// TwinCAT 3 PLC project PLC
// ProgramVersion: 3.1.4022.1
// libraries:
//   Tc2_Standard, * (Beckhoff Automation GmbH)
//   Tc2_System, * (Beckhoff Automation GmbH)
//   Tc3_EventLogger, * (Beckhoff Automation GmbH)
//   Tc3_Module, * (Beckhoff Automation GmbH)
//   Tc3_JsonXml,3.3.4.0,Beckhoff Automation GmbH
// project tree:
//   DUTs/ ST_AI.TcDUT, ST_Led.TcDUT, ST_Values_LineChart.TcDUT
//   / GlobalTextList.TcGTLO, PlcTask.TcTTO
//   GVLs/ HMI.TcGVL
//   POUs/ CHART.TcPOU, FB_Blink.TcPOU, FB_LineChart.TcPOU, MAIN.TcPOU, SCOPE.TcPOU
//   POUs/Motor/ FB_Motor.TcPOU, ST_MotorParam.TcDUT
//   POUs/Valve/ FB_Valve.TcPOU, ST_ValveParam.TcDUT
// real-time tasks:
//   TASK PlcTask: cycle T#10ms, priority 20, ADS port 350

CONFIGURATION PLC
    RESOURCE PLC ON TwinCAT3
        TASK PlcTask(INTERVAL := T#10ms, PRIORITY := 20);
        PROGRAM MAIN WITH PlcTask : MAIN;
    END_RESOURCE
END_CONFIGURATION

// ---- DUTs/ST_AI.TcDUT
TYPE ST_AI :
STRUCT
ID: STRING;
Measure:REAL;
Low_Range:REAL;
High_Range:REAL;
Decimals:INT;
Unit:STRING;
Alarmtype:INT;
LowLimit: REAL;
LowDelay:DINT;
LowAlarm:BOOL;
HighLimit: REAL;
HighDelay:DINT;
HighAlarm:BOOL;
Sensortype:INT;
ShortCircuitAlarm:BOOL;
BrokenWireAlarm:BOOL;
Offset:REAL;
ManualValue:REAL;
ManualControl:INT;
END_STRUCT
END_TYPE

// ---- DUTs/ST_Led.TcDUT
TYPE ST_Led :
STRUCT
	sName 		: STRING;
	bControl	: BOOL;
	bStatus 	: BOOL;
	nValue		: REAL;
END_STRUCT
END_TYPE

// ---- DUTs/ST_Values_LineChart.TcDUT
TYPE ST_Values_LineChart :
STRUCT
	x:LREAL;
	y:LREAL;

END_STRUCT
END_TYPE

// ---- POUs/Motor/ST_MotorParam.TcDUT
TYPE ST_MotorParam :
STRUCT
	Unit : STRING;
	Set : INT;
	P: UINT;
	I: UINT;
	D: UINT;
END_STRUCT
END_TYPE

// ---- POUs/Valve/ST_ValveParam.TcDUT
TYPE ST_ValveParam :
STRUCT
	Unit : STRING;
	Set : INT;
	P: UINT;
	I: UINT;
	D: UINT;
END_STRUCT
END_TYPE

// ---- GVLs/HMI.TcGVL
{attribute 'qualified_only'}
VAR_GLOBAL
	bEnableLed	: BOOL;
	bLedStatus	: BOOL;
	stAi		: ST_AI;
	arrStLeds	: ARRAY[1..NUM_OF_LEDS] OF ST_Led := 
	[
		(sName := 'Led #01'),
		(sName := 'Led #02'),
		(sName := 'Led #03'),
		(sName := 'Led #04'),
		(sName := 'Led #05'),
		(sName := 'Led #06'),
		(sName := 'Led #07'),
		(sName := 'Led #08'),
		(sName := 'Led #09'),
		(sName := 'Led #10')
	];
	arrPersons	: ARRAY [1..NUM_OF_PERSONS] OF STRING := 
	[
		'Person1',
		'Person2',
		'Person3',
		'Person4',
		'Person5',
		'Person6',
		'Person7',
		'Person8',
		'Person9',
		'Person10'
	];
	SineVerySlow	: LREAL;
END_VAR

VAR_GLOBAL CONSTANT
	NUM_OF_LEDS : INT := 10;	
	NUM_OF_PERSONS : INT := 10;
END_VAR

// ---- POUs/MAIN.TcPOU
PROGRAM MAIN
VAR
	fbBlink		: FB_Blink;
	arrFbBlink 	: ARRAY [1..HMI.NUM_OF_LEDS] OF FB_Blink;
	i: INT;
	a: INT;
	b: INT := 1000;
	asdf: INT;
	stAi: INT;
	adfsaa: UINT;
	bInitAlarms: BOOL;
	sString : STRING := '{"color": "rgba(255,191,127,1)"}';
	
	fbEventLogger : FB_TcEventLogger;
	fbAlarm01 : FB_TcAlarm;
	fbMessage01 : FB_TcMessage;
	bTriggerAlarm01 : BOOL;
	bConfirmAlarm01 : BOOL;
	bClearAlarm01	: BOOL;
	
	stLed : REFERENCE TO ST_LED;
	stLedInstance : ST_LED;
	
	fbValve: FB_Valve;
	fbMotor: FB_Motor;
	LOGSTUFF: BOOL;
	asd: DINT;
END_VAR


// Yksittäisen FB:n kutsuminen
fbBlink(
	i_bEnable:= HMI.bEnableLed, 
	i_tTime := T#1S, 
	O_bOut=> hmi.bLedStatus
); 

// Taulukossa olevien FB:iden kutsuminen
FOR i := 1 TO HMI.NUM_OF_LEDS DO
	arrFbBlink[i]
	(
		i_sName 	:= HMI.arrStLeds[i].sName,
		i_bEnable 	:= HMI.arrStLeds[i].bControl,
		o_bOut		=> HMI.arrStLeds[i].bStatus
	);
END_FOR

SCOPE();

asdf := SIZEOF(HMI.stAi);
adfsaa := SIZEOF(HMI.arrStLeds[1]);


IF (NOT bInitAlarms) THEN
	bInitAlarms:=TRUE;
	fbAlarm01.CreateEx(TC_EVENTS.AlarmsClass.Alarm01,TRUE,0);
	fbMessage01.CreateEx(TC_EVENTS.AlarmsClass.Message01, 0);
END_IF

IF (bTriggerAlarm01) THEN
	fbAlarm01.Raise(0);
	bTriggerAlarm01 := FALSE;
END_IF

IF (bConfirmAlarm01) THEN
	fbAlarm01.Confirm(0);
	bConfirmAlarm01:= FALSE;
END_IF

IF (bClearAlarm01) THEN
	fbAlarm01.Clear(0,TRUE);
	bClearAlarm01 := FALSE;
	fbMessage01.Send(0);
END_IF

stLedInstance.nValue:=100;
stLed REF=stLedInstance;

fbValve();
fbMotor();

IF LOGSTUFF AND a<b THEN
	fbMessage01.ipArguments.Clear();
	fbMessage01.ipArguments.AddDInt(a);
	fbMessage01.Send(0);
	a:=a+1;
END_IF

END_PROGRAM

// ---- POUs/FB_Blink.TcPOU
FUNCTION_BLOCK FB_Blink
VAR_INPUT
	i_sName	: STRING;
	i_bEnable: BOOL;
	i_tTime: TIME := T#1S;
END_VAR
VAR_OUTPUT
	o_bOut: BOOL;
END_VAR
VAR
	T1_TON: TON;
	T2_TOF: TOF;
END_VAR

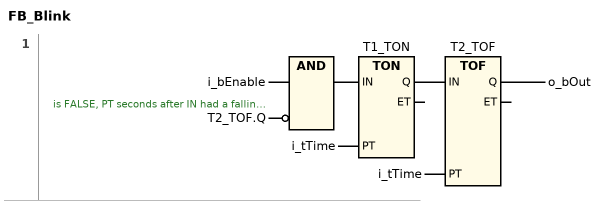
// NETWORK 1
//   T2_TOF.Q: is FALSE, PT seconds after IN had a falling edge
T1_TON(IN := i_bEnable AND NOT T2_TOF.Q, PT := i_tTime); // TON
T2_TOF(IN := T1_TON.Q, PT := i_tTime); // TOF
o_bOut := T2_TOF.Q;

END_FUNCTION_BLOCK

// ---- POUs/Valve/FB_Valve.TcPOU
FUNCTION_BLOCK FB_Valve
VAR_INPUT
END_VAR
VAR_OUTPUT
END_VAR
VAR
	Value 		: LREAL;
	Parameters 	: ST_ValveParam := (Set := 1, P := 2, I := 3, D := 4, Unit:='Deg');
END_VAR

Value := HMI.SineVerySlow*180/2;

END_FUNCTION_BLOCK

// ---- POUs/Motor/FB_Motor.TcPOU
FUNCTION_BLOCK FB_Motor
VAR_INPUT
END_VAR
VAR_OUTPUT
END_VAR
VAR
	Value 		: LREAL;
	Parameters 	: ST_MotorParam := (Set := 1, P := 2, I := 3, D := 4, Unit:='%');
END_VAR

Value := HMI.SineVerySlow*100/2;

METHOD Start : BOOL
VAR_INPUT
END_VAR
END_METHOD

END_FUNCTION_BLOCK

// ---- POUs/SCOPE.TcPOU
PROGRAM SCOPE
VAR
	i				: UINT;
	j				: UINT:=1;
	t				: UINT;
	
	Cosinus_Half	: LREAL;
	Sinus_Fast		: LREAL;
	Sinus_Fast50	: LREAL;
	Sinus_Slow20	: LREAL;
	Sinus_Slow1		: LREAL;
	Sinus_Slow2		: LREAL;
	Sinus_VerySlow	: LREAL;
	Sinus_SqFast	: LREAL;
	Sinus_SqSlow	: REAL;
	Sinus_Cos_Half	: LREAL;
	SinglePeak		: LREAL;
	phi				: REAL;
	Ts				: UINT;
	vs: LREAL;
	t2: LREAL;
	(* Histogram *)
	arrHistogramData: ARRAY[0..NUM_OF_ROWS] OF LREAL;
	fTimeStep	: LREAL := 0.001;
	omega_t		: ARRAY[0..NUM_OF_ROWS] OF LREAL;

	fTemp		: LREAL;
	ii: INT;
	bInit: BOOL := true;
	fStep: LREAL;
END_VAR

VAR_TEMP
	Cosinus_Fast: LREAL;
END_VAR

VAR CONSTANT
	NUM_OF_ROWS: INT := 99;
END_VAR


	
	vs := vs + 0.001;
	t := t + 1;
	t2 := t2 + 1.05;
	i:=i+1;
	Ts:=128*10;
	SinglePeak:=0;
	
	IF (t>=2*Ts) THEN
		j:=j+1;
		t:=t-2*Ts;
	END_IF
	
	phi:=t/Ts;
	Cosinus_Half:=COS(PI*t/(2*Ts));
	HMI.SineVerySlow := Sinus_VerySlow:=1 + SIN(vs);
	Sinus_Slow1:=COS(4*PI* (t+Ts/4+phi)/Ts);
	Sinus_Slow20 := 15 + 5 * Sinus_Slow1;
	Sinus_Slow2:= Sinus_VerySlow*COS(4*PI* (t+Ts/3+phi)/Ts);
	Sinus_Fast:=COS(12*PI*t/Ts);
	Sinus_Fast50:=50 + 50* SIN(6*PI*t/Ts);
	Cosinus_Fast:=SIN(12*PI*t2/Ts);
	Sinus_SqFast:=Sinus_Fast* Sinus_Slow1;
	Sinus_SqSlow:=LREAL_TO_REAL(Sinus_VerySlow*Sinus_Slow1);
	
(**** Histogram ***********************)

IF bInit THEN
	fStep := 2*PI/(NUM_OF_ROWS+1);
	FOR ii := 1 TO NUM_OF_ROWS DO
		omega_t[ii] := omega_t[ii-1] + SIN(fStep);
	END_FOR
	bInit:= FALSE;
END_IF

FOR ii := 0 TO NUM_OF_ROWS DO
	omega_t[ii] := omega_t[ii] + fTimeStep;
	fTemp := 20 * SIN(omega_t[ii]);
	arrHistogramData[ii] := fTemp;
END_FOR

END_PROGRAM

// ---- POUs/CHART.TcPOU
PROGRAM CHART
VAR
	arrChartData : ARRAY[0..1,0..199] OF ST_Values_LineChart;
	bEnable: BOOL := true;
	fbLineChart: FB_LineChart;
END_VAR


fbLineChart(
	i_bEnable			:= bEnable := TRUE, 
	i_tUpdateInterval	:= T#100MS, 
	i_fCh1Value			:= SCOPE.Sinus_Fast50, 
	i_fCh2Value			:= SCOPE.Sinus_Slow20, 
	arrChartData		:= arrChartData
);

END_PROGRAM

// ---- POUs/FB_LineChart.TcPOU
FUNCTION_BLOCK FB_LineChart
VAR_INPUT
	i_bEnable : BOOL;
	i_tUpdateInterval : TIME := T#100MS;
	i_fCh1Value : LREAL;
	i_fCh2Value	: LREAL;
	
END_VAR
VAR_OUTPUT
END_VAR
VAR_IN_OUT
	arrChartData : ARRAY[0..1,0..199] OF ST_Values_LineChart;
END_VAR
VAR
	i: INT;
	str: STRING;
	bTick: BOOL;
	bReset: BOOL := TRUE;
	T1_TON: Ton;
	nStep: REAL := 0.25;	
END_VAR



T1_TON(IN := NOT T1_TON.Q AND i_bEnable, PT := i_tUpdateInterval, Q=>bTick);

IF bTick THEN
	
   FOR i := 198 TO 0 BY -1 DO
	   arrChartData[0,i+1].y := arrChartData[0,i].y; 
	   arrChartData[1,i+1].y := arrChartData[1,i].y; 
   END_FOR
   
   arrChartData[0,0].y := i_fCh1Value;
   arrChartData[1,0].y := i_fCh2Value;
   
END_IF

IF bReset THEN 
	
	FOR i:=0 TO 199 BY 1 DO
	   arrChartData[0,i].x := i * nStep;
	   arrChartData[0,i].y := 0;
	   arrChartData[1,i].x := i * nStep;
	   arrChartData[1,i].y := 0;
	END_FOR
	
	bReset := FALSE;
	
END_IF

END_FUNCTION_BLOCK
